# EPICS StreamDevice protocol: thorlabs/dualslider/dualslider.proto
#thorlabs
Terminator = CR LF;

debug{
    out "%s";
    in "%39c";
}

id{
    out "0in";
    in "%39c";
    @init{out "0in";in "%39c";}
}

gs{
    out "0gs";
    in "0GS%2d";
    @init{out "0gs";in "0GS%2d";}
}

gp{
    out "0gp";
    in "0PO%{00000000|0000001F}";
    @init{out "0gp";in "0PO%x";}
}

pos_set{
    out "0%{bw|fw}";
    in "0%{GS|PO}%x";
    @init{gp;}

}

#fw{
#    out "0fw";
#    in "0%{GS|PO}%d";
#    @init{gp;}
#}
#
#
#bw{
#    out "0bw";
#    in "0%{GS|PO}%d";
#    @init{gp;}
#}
